FUNCTION_BLOCK HMI_EM_Template_Gain EXTENDS FB_HMI_Base
VAR_INPUT
END_VAR
VAR_OUTPUT
END_VAR
VAR
	s_itfEmTemplate			: ITF_EM_Template; // Upgraded Interface from Control module
// Hmi Control Modules 
	// n.a.
// Hmi Alarms
	// n.a.
// Local vars
	// n.a.
	
END_VAR

SUPER^();

METHOD PUBLIC m_Main
SUPER^.m_Main();


// Upgrade the base-interface
IF NOT __QUERYINTERFACE(i_itfModule, s_itfEmTemplate) THEN
	RETURN;
END_IF

// Sub EMs
	// n.a.

// Control modules
	// CM_....
	// n.a.
END_METHOD

END_FUNCTION_BLOCK

(* stored: Version 1.1.0.1, ProductVersion 3.1.4024.10
   POU HMI_EM_Template_Gain: Id {ee1a0384-e929-4b85-8e7a-f49b8c162404}, SpecialFunc None
   Method m_Main: Id {de5865cd-34bc-46d4-874e-7964e72958e8} *)
